// TIA Portal V16 export
// export: Created 2021-05-25T16:14:39.8533529Z, ExportSetting WithDefaults, DisplayName Totally Integrated Automation Portal, DisplayVersion V16, DisplayName TIA Portal Version Control Interface, DisplayVersion V16, DisplayName TIA Portal Openness, DisplayVersion V16, DisplayName STEP 7 Professional, DisplayVersion V16, DisplayName STEP 7 Safety, DisplayVersion V16, DisplayName WinCC Unified SCADA Engineering System, DisplayVersion V16
DATA_BLOCK "dbDO"   // DB11
{ S7_Optimized_Access := 'FALSE'; DB_Accessible_From_OPC_UA := 'FALSE' }
VERSION : 0.1
// stored: AutoNumber false, DBAccessibleFromOPCUA false, IsOnlyStoredInLoadMemory false, IsWriteProtectedInAS false
   VAR
      SEMAFOR_ZELENA : Bool;
      SEMAFOR_RUMENA : Bool;
      SEMAFOR_RDECA : Bool;
      Spare0_3 { ExternalAccessible := 'False'; ExternalVisible := 'False'; ExternalWritable := 'False'} : Bool;
      Spare0_4 { ExternalAccessible := 'False'; ExternalVisible := 'False'; ExternalWritable := 'False'} : Bool;
      Spare0_5 { ExternalAccessible := 'False'; ExternalVisible := 'False'; ExternalWritable := 'False'} : Bool;
      Spare0_6 { ExternalAccessible := 'False'; ExternalVisible := 'False'; ExternalWritable := 'False'} : Bool;
      Spare0_7 { ExternalAccessible := 'False'; ExternalVisible := 'False'; ExternalWritable := 'False'} : Bool;
      Spare1_0 { ExternalAccessible := 'False'; ExternalVisible := 'False'; ExternalWritable := 'False'} : Bool;
      Spare1_1 { ExternalAccessible := 'False'; ExternalVisible := 'False'; ExternalWritable := 'False'} : Bool;
      Spare1_2 { ExternalAccessible := 'False'; ExternalVisible := 'False'; ExternalWritable := 'False'} : Bool;
      Spare1_3 { ExternalAccessible := 'False'; ExternalVisible := 'False'; ExternalWritable := 'False'} : Bool;
      Spare1_4 { ExternalAccessible := 'False'; ExternalVisible := 'False'; ExternalWritable := 'False'} : Bool;
      Spare1_5 { ExternalAccessible := 'False'; ExternalVisible := 'False'; ExternalWritable := 'False'} : Bool;
      Spare1_6 { ExternalAccessible := 'False'; ExternalVisible := 'False'; ExternalWritable := 'False'} : Bool;
      Spare1_7 { ExternalAccessible := 'False'; ExternalVisible := 'False'; ExternalWritable := 'False'} : Bool;
      VKLOP_M_TRACNEGA_TRANS_NOGIC : Bool;   // (Q0.0)
      VKLOP_VIBRATORJA : Bool;   // (Q0.1)
      VKLOP_M_TRAKA_VIJACNIKA : Bool;   // (Q0.2)
      Spare20_3 { ExternalAccessible := 'False'; ExternalVisible := 'False'; ExternalWritable := 'False'} : Bool;
      Spare20_4 { ExternalAccessible := 'False'; ExternalVisible := 'False'; ExternalWritable := 'False'} : Bool;
      Spare20_5 { ExternalAccessible := 'False'; ExternalVisible := 'False'; ExternalWritable := 'False'} : Bool;
      Spare20_6 { ExternalAccessible := 'False'; ExternalVisible := 'False'; ExternalWritable := 'False'} : Bool;
      Spare20_7 { ExternalAccessible := 'False'; ExternalVisible := 'False'; ExternalWritable := 'False'} : Bool;
      MOTOR_1_ZADAJ_DESNO_START : Bool;   // (Q1.1)
      MOTOR_1_ZADAJ_DESNO_RESET : Bool;   // (Q1.2)
      MOTOR_1_ZADAJ_DESNO_HITROST : Bool;   // (Q1.3)
      MOTOR_1_ZADAJ_DESNO_SMER : Bool;   // (Q1.4)
      MOTOR_2_SPREDAJ_DESNO_START : Bool;   // (Q1.5)
      MOTOR_2_SPREDAJ_DESNO_RESET : Bool;   // (Q1.6)
      MOTOR_2_SPREDAJ_DESNO_HITROST : Bool;   // (Q1.7)
      MOTOR_2_SPREDAJ_DESNO_SMER : Bool;
      MOTOR_1_ZADAJ_LEVO_START : Bool;
      MOTOR_1_ZADAJ_LEVO_RESET : Bool;
      MOTOR_1_ZADAJ_LEVO_HITROST : Bool;
      MOTOR_1_ZADAJ_LEVO_SMER : Bool;
      MOTOR_2_SPREDAJ_LEVO_START : Bool;
      MOTOR_2_SPREDAJ_LEVO_RESET : Bool;
      MOTOR_2_SPREDAJ_LEVO_HITROST : Bool;
      MOTOR_2_SPREDAJ_LEVO_SMER : Bool;
      Spare23_0 { ExternalAccessible := 'False'; ExternalVisible := 'False'; ExternalWritable := 'False'} : Bool;
      Spare23_1 { ExternalAccessible := 'False'; ExternalVisible := 'False'; ExternalWritable := 'False'} : Bool;
      Spare23_2 { ExternalAccessible := 'False'; ExternalVisible := 'False'; ExternalWritable := 'False'} : Bool;
      Spare23_3 { ExternalAccessible := 'False'; ExternalVisible := 'False'; ExternalWritable := 'False'} : Bool;
      Spare23_4 { ExternalAccessible := 'False'; ExternalVisible := 'False'; ExternalWritable := 'False'} : Bool;
      Spare23_5 { ExternalAccessible := 'False'; ExternalVisible := 'False'; ExternalWritable := 'False'} : Bool;
      Spare23_6 { ExternalAccessible := 'False'; ExternalVisible := 'False'; ExternalWritable := 'False'} : Bool;
      Spare23_7 { ExternalAccessible := 'False'; ExternalVisible := 'False'; ExternalWritable := 'False'} : Bool;
   END_VAR
BEGIN
END_DATA_BLOCK
